(* IEC 61131-3 sources: Lasal/CPU_5344_V01/Class/generalMPScontrolSettings, 1 file *)

(* ---- generalMPScontrolSettings.st ---- *)
(*!
<Class
	Name               = "generalMPScontrolSettings"
	Revision           = "1.0"
	RealtimeTask       = "false"
	CyclicTask         = "false"
	BackgroundTask     = "false"
	Sigmatek           = "false"
	OSInterface        = "false"
	HighPriority       = "false"
	Automatic          = "false"
	UpdateMode         = "Prescan"
	SharedCommandTable = "true"
	Objectsize         = "(660,1080)">
	<Channels>
		<Server Name="addOutputOperations" Visualized="true" Initialize="true" WriteProtected="false" Retentive="false"/>
		<Server Name="amountOfUnits" Visualized="true" Initialize="true" DefValue="7" WriteProtected="false" Retentive="false"/>
		<Server Name="ClassSvr" Visualized="false" Initialize="false" WriteProtected="true" Retentive="false"/>
		<Server Name="combineOperations" Visualized="true" Initialize="true" DefValue="1" WriteProtected="false" Retentive="false"/>
		<Server Name="freeLoadDistance" Visualized="true" Initialize="false" WriteProtected="false" Retentive="false"/>
		<Server Name="gripDistanceInputWagon" Visualized="true" Initialize="false" WriteProtected="false" Retentive="false"/>
		<Server Name="lengthBetweenPieces" Visualized="true" Initialize="false" WriteProtected="false" Retentive="false"/>
		<Server Name="machineName" Class="StringRAM" Visualized="true" Remotely="true" Initialize="true" WriteProtected="false" Retentive="false"/>
		<Server Name="maxProductLength" Visualized="true" Initialize="true" WriteProtected="false" Retentive="false"/>
		<Server Name="maxScrapLength" Visualized="true" Initialize="false" WriteProtected="false" Retentive="false"/>
		<Server Name="maxTakeOverPos" Visualized="true" Initialize="false" WriteProtected="false" Retentive="false"/>
		<Server Name="minPosWagonUp" Visualized="true" Initialize="false" WriteProtected="false" Retentive="false"/>
		<Server Name="minProductLength" Visualized="true" Initialize="true" DefValue="1000" WriteProtected="false" Retentive="false"/>
		<Server Name="minScrapLengthEnd" Visualized="true" Initialize="false" WriteProtected="false" Retentive="false"/>
		<Server Name="minScrapLengthFront" Visualized="true" Initialize="false" WriteProtected="false" Retentive="false"/>
		<Server Name="minTakeOverPos" Visualized="true" Initialize="false" WriteProtected="false" Retentive="false"/>
		<Server Name="moveBigWasteToMagazine" Visualized="true" Initialize="false" WriteProtected="true" Retentive="false"/>
		<Server Name="moveToMinPosAfterProduction" Visualized="true" Initialize="true" DefValue="0" WriteProtected="false" Retentive="false"/>
		<Server Name="MPS_nr" Visualized="true" Initialize="true" DefValue="4444" WriteProtected="true" Retentive="false"/>
		<Server Name="noEndSaw" Visualized="true" Initialize="false" WriteProtected="false" Retentive="false"/>
		<Server Name="noFrontSaw" Visualized="true" Initialize="false" WriteProtected="false" Retentive="false"/>
		<Server Name="noWasteStop" Visualized="true" Initialize="false" WriteProtected="false" Retentive="false"/>
		<Server Name="optimumTakeOverPos" Visualized="true" Initialize="false" WriteProtected="false" Retentive="false"/>
		<Server Name="overtakeActive" Visualized="true" Initialize="false" WriteProtected="false" Retentive="false"/>
		<Server Name="turnPointSawAtOutputSide" Visualized="true" Initialize="false" WriteProtected="false" Retentive="false"/>
		<Server Name="wasteAtFront" Visualized="true" Initialize="false" WriteProtected="false" Retentive="false"/>
		<Server Name="wasteStopForEndWaste" Visualized="true" Initialize="false" WriteProtected="false" Retentive="false"/>
		<Server Name="yPosTurnPointSaw" Visualized="true" Initialize="false" WriteProtected="false" Retentive="false"/>
		<Client Name="ctrlCalc" Required="true" Internal="false"/>
		<Client Name="ctrlSettings" Required="true" Internal="false"/>
		<Client Name="iMaxPosWagon" Required="true" Internal="false"/>
		<Client Name="typeMachine" Required="true" Internal="true"/>
	</Channels>
	<Network Name="generalMPScontrolSettings">
		<!-- List of Components in this network -->
		<Components>
			<Object
				Name       = "typeMachine"
				Class      = "StringRAM"
				Position   = "(60,180)"
				Visualized = "true"
				Remotely   = "true">
				<Channels>
					<Server Name="Data"/>
					<Client Name="SingleRealloc" Value="1"/>
					<Client Name="UseFile"/>
				</Channels>
			</Object>
		</Components>
		<Comments>
		</Comments>
		<!-- List of Connections in this network -->
		<Connections>
			<Connection Source="this.typeMachine" Destination="typeMachine.Data"/>
			<Connection Source="this.machineName" Destination="typeMachine.Data" Vertices="(758,330),(586,270),"/>
		</Connections>
		<!-- Headerfiles -->
		<Options>
		</Options>
	</Network>
</Class>
*)
generalMPScontrolSettings : CLASS
  //Servers:
	ClassSvr 	: SvrChCmd_DINT;
	MPS_nr 	: SvrCh_DINT;
	machineName 	: SvrChCmd_UDINT;
	amountOfUnits 	: SvrCh_DINT;
	minProductLength 	: SvrCh_DINT;
	maxProductLength 	: SvrCh_DINT;
	minScrapLengthFront 	: SvrCh_DINT;
	minScrapLengthEnd 	: SvrCh_DINT;
	maxScrapLength 	: SvrCh_DINT;
	lengthBetweenPieces 	: SvrCh_DINT;
	freeLoadDistance 	: SvrCh_DINT;
	noFrontSaw 	: SvrCh_DINT;
	noEndSaw 	: SvrCh_DINT;
	wasteAtFront 	: SvrCh_DINT;
	turnPointSawAtOutputSide 	: SvrCh_DINT;
	yPosTurnPointSaw 	: SvrCh_DINT;
	moveToMinPosAfterProduction 	: SvrCh_DINT;
	gripDistanceInputWagon 	: SvrCh_DINT;
	moveBigWasteToMagazine 	: SvrCh_DINT;
	overtakeActive 	: SvrCh_DINT;
	combineOperations 	: SvrCh_DINT;
	noWasteStop 	: SvrCh_DINT;
	wasteStopForEndWaste 	: SvrCh_DINT;
	optimumTakeOverPos 	: SvrCh_DINT;
	minTakeOverPos 	: SvrCh_DINT;
	maxTakeOverPos 	: SvrCh_DINT;
	minPosWagonUp 	: SvrCh_DINT;
	addOutputOperations 	: SvrCh_DINT;
  //Clients:
	typeMachine 	: CltChCmd_StringRAM;
	ctrlSettings 	: CltChCmd_dbSettings;
	iMaxPosWagon 	: CltCh_DINT;
	ctrlCalc 	: CltChCmd_calcOperationListV2;
  //Variables:
  //Functions:

	FUNCTION VIRTUAL GLOBAL machineName::Read
		VAR_OUTPUT
			output (EAX) 	: UDINT;
		END_VAR;

	FUNCTION VIRTUAL GLOBAL machineName::Write
		VAR_INPUT
			input (EAX) 	: UDINT;
		END_VAR
		VAR_OUTPUT
			result (EAX) 	: UDINT;
		END_VAR;

	FUNCTION VIRTUAL GLOBAL maxProductLength::Read
		VAR_OUTPUT
			output (EAX) 	: DINT;
		END_VAR;

	FUNCTION VIRTUAL GLOBAL maxProductLength::Write
		VAR_INPUT
			input (EAX) 	: DINT;
		END_VAR
		VAR_OUTPUT
			result (EAX) 	: DINT;
		END_VAR;

	FUNCTION VIRTUAL GLOBAL minScrapLengthFront::Read
		VAR_OUTPUT
			output (EAX) 	: DINT;
		END_VAR;

	FUNCTION VIRTUAL GLOBAL minScrapLengthEnd::Read
		VAR_OUTPUT
			output (EAX) 	: DINT;
		END_VAR;

	FUNCTION VIRTUAL GLOBAL maxScrapLength::Read
		VAR_OUTPUT
			output (EAX) 	: DINT;
		END_VAR;

	FUNCTION VIRTUAL GLOBAL lengthBetweenPieces::Read
		VAR_OUTPUT
			output (EAX) 	: DINT;
		END_VAR;

	FUNCTION VIRTUAL GLOBAL freeLoadDistance::Read
		VAR_OUTPUT
			output (EAX) 	: DINT;
		END_VAR;

	FUNCTION VIRTUAL GLOBAL noFrontSaw::Read
		VAR_OUTPUT
			output (EAX) 	: DINT;
		END_VAR;

	FUNCTION VIRTUAL GLOBAL noEndSaw::Read
		VAR_OUTPUT
			output (EAX) 	: DINT;
		END_VAR;

	FUNCTION VIRTUAL GLOBAL wasteAtFront::Read
		VAR_OUTPUT
			output (EAX) 	: DINT;
		END_VAR;

	FUNCTION VIRTUAL GLOBAL turnPointSawAtOutputSide::Read
		VAR_OUTPUT
			output (EAX) 	: DINT;
		END_VAR;

	FUNCTION VIRTUAL GLOBAL yPosTurnPointSaw::Read
		VAR_OUTPUT
			output (EAX) 	: DINT;
		END_VAR;

	FUNCTION VIRTUAL GLOBAL moveToMinPosAfterProduction::Read
		VAR_OUTPUT
			output (EAX) 	: DINT;
		END_VAR;

	FUNCTION VIRTUAL GLOBAL gripDistanceInputWagon::Read
		VAR_OUTPUT
			output (EAX) 	: DINT;
		END_VAR;

	FUNCTION VIRTUAL GLOBAL moveBigWasteToMagazine::Read
		VAR_OUTPUT
			output (EAX) 	: DINT;
		END_VAR;

	FUNCTION VIRTUAL GLOBAL overtakeActive::Read
		VAR_OUTPUT
			output (EAX) 	: DINT;
		END_VAR;

	FUNCTION VIRTUAL GLOBAL noWasteStop::Read
		VAR_OUTPUT
			output (EAX) 	: DINT;
		END_VAR;

	FUNCTION VIRTUAL GLOBAL wasteStopForEndWaste::Read
		VAR_OUTPUT
			output (EAX) 	: DINT;
		END_VAR;

	FUNCTION VIRTUAL GLOBAL optimumTakeOverPos::Read
		VAR_OUTPUT
			output (EAX) 	: DINT;
		END_VAR;

	FUNCTION VIRTUAL GLOBAL minTakeOverPos::Read
		VAR_OUTPUT
			output (EAX) 	: DINT;
		END_VAR;

	FUNCTION VIRTUAL GLOBAL maxTakeOverPos::Read
		VAR_OUTPUT
			output (EAX) 	: DINT;
		END_VAR;

	FUNCTION VIRTUAL GLOBAL minPosWagonUp::Read
		VAR_OUTPUT
			output (EAX) 	: DINT;
		END_VAR;
  //Tables:
	FUNCTION @STD
		VAR_OUTPUT
			ret_code	: CONFSTATES;
		END_VAR;
	FUNCTION GLOBAL TAB @CT_;
END_CLASS;

#pragma using StringRAM
#pragma usingLtd calcOperationListV2
#pragma usingLtd dbSettings

// JdK 4-2-2020: generalMPScontrolSettings created for first test to read in settings to pc
// at this moment the class is only for storage off fixed machine data

FUNCTION VIRTUAL GLOBAL generalMPScontrolSettings::machineName::Read
	VAR_OUTPUT
		output (EAX) 	: UDINT;
	END_VAR

	machineName := typeMachine.Data.Read();
	output := machineName;

END_FUNCTION

FUNCTION VIRTUAL GLOBAL generalMPScontrolSettings::machineName::Write
	VAR_INPUT
		input (EAX) 	: UDINT;
	END_VAR
	VAR_OUTPUT
		result (EAX) 	: UDINT;
	END_VAR

	machineName := input;
	result := (typeMachine.Data.Write(machineName))$UDINT;

END_FUNCTION

FUNCTION VIRTUAL GLOBAL generalMPScontrolSettings::maxProductLength::Read
	VAR_OUTPUT
		output (EAX) 	: DINT;
	END_VAR

  iMaxPosWagon:= iMaxPosWagon.Read();
  maxProductLength:=iMaxPosWagon-ctrlSettings.offsetTakeIn-ctrlSettings.freeSpaceLoadMaterial;
	output := maxProductLength;

END_FUNCTION

FUNCTION VIRTUAL GLOBAL generalMPScontrolSettings::minScrapLengthFront::Read
	VAR_OUTPUT
		output (EAX) 	: DINT;
	END_VAR
  minScrapLengthFront:=ctrlSettings.minFrontWaste;
	output := minScrapLengthFront;

END_FUNCTION

FUNCTION VIRTUAL GLOBAL generalMPScontrolSettings::minScrapLengthEnd::Read
	VAR_OUTPUT
		output (EAX) 	: DINT;
	END_VAR
  minScrapLengthEnd:=ctrlSettings.minEndWaste;
	output := minScrapLengthEnd;

END_FUNCTION

FUNCTION VIRTUAL GLOBAL generalMPScontrolSettings::maxScrapLength::Read
	VAR_OUTPUT
		output (EAX) 	: DINT;
	END_VAR
  maxScrapLength:=ctrlSettings.maxLengthWaste;
	output := maxScrapLength;

END_FUNCTION

FUNCTION VIRTUAL GLOBAL generalMPScontrolSettings::freeLoadDistance::Read
	VAR_OUTPUT
		output (EAX) 	: DINT;
	END_VAR
  freeLoadDistance:=ctrlSettings.freeSpaceLoadMaterial;
	output := freeLoadDistance;

END_FUNCTION

FUNCTION VIRTUAL GLOBAL generalMPScontrolSettings::noFrontSaw::Read
	VAR_OUTPUT
		output (EAX) 	: DINT;
	END_VAR
  noFrontSaw:=ctrlSettings.doFrontWaste=0;//   .DoFrontWastePiece=0;
	output := noFrontSaw;

END_FUNCTION

FUNCTION VIRTUAL GLOBAL generalMPScontrolSettings::noEndSaw::Read
	VAR_OUTPUT
		output (EAX) 	: DINT;
	END_VAR
  noEndSaw:=ctrlSettings.DoEndWaste=0;
	output := noEndSaw;

END_FUNCTION

FUNCTION VIRTUAL GLOBAL generalMPScontrolSettings::wasteAtFront::Read
	VAR_OUTPUT
		output (EAX) 	: DINT;
	END_VAR
  wasteAtFront:=ctrlSettings.allWasteAtFront;
	output := wasteAtFront;

END_FUNCTION

FUNCTION VIRTUAL GLOBAL generalMPScontrolSettings::turnPointSawAtOutputSide::Read
	VAR_OUTPUT
		output (EAX) 	: DINT;
	END_VAR
  turnPointSawAtOutputSide:=ctrlCalc.sParTurnPointAtOutputSide;
	output := turnPointSawAtOutputSide;

END_FUNCTION

FUNCTION VIRTUAL GLOBAL generalMPScontrolSettings::yPosTurnPointSaw::Read
	VAR_OUTPUT
		output (EAX) 	: DINT;
	END_VAR
  yPosTurnPointSaw:=ctrlCalc.sParYposTurnPoint;
	output := yPosTurnPointSaw;

END_FUNCTION

FUNCTION VIRTUAL GLOBAL generalMPScontrolSettings::moveToMinPosAfterProduction::Read
	VAR_OUTPUT
		output (EAX) 	: DINT;
	END_VAR
  moveToMinPosAfterProduction:=ctrlCalc;
	output := moveToMinPosAfterProduction;

END_FUNCTION

FUNCTION VIRTUAL GLOBAL generalMPScontrolSettings::gripDistanceInputWagon::Read
	VAR_OUTPUT
		output (EAX) 	: DINT;
	END_VAR
  gripDistanceInputWagon:=ctrlSettings.lengthGripProfile;
	output := gripDistanceInputWagon;

END_FUNCTION

FUNCTION VIRTUAL GLOBAL generalMPScontrolSettings::moveBigWasteToMagazine::Read
	VAR_OUTPUT
		output (EAX) 	: DINT;
	END_VAR

  moveBigWasteToMagazine:= ctrlSettings.moveBigWasteToMagazin;
	output := moveBigWasteToMagazine;

END_FUNCTION

FUNCTION VIRTUAL GLOBAL generalMPScontrolSettings::overtakeActive::Read
	VAR_OUTPUT
		output (EAX) 	: DINT;
	END_VAR

  overtakeActive:= ctrlSettings.overTakeActive;
	output := overtakeActive;

END_FUNCTION

FUNCTION VIRTUAL GLOBAL generalMPScontrolSettings::noWasteStop::Read
	VAR_OUTPUT
		output (EAX) 	: DINT;
	END_VAR

  noWasteStop:= ctrlSettings.noWasteStop;
	output := noWasteStop;

END_FUNCTION

FUNCTION VIRTUAL GLOBAL generalMPScontrolSettings::wasteStopForEndWaste::Read
	VAR_OUTPUT
		output (EAX) 	: DINT;
	END_VAR

  wasteStopForEndWaste:= ctrlSettings.wasteStopForEndWaste & ctrlSettings.noWasteStop=0;
	output := wasteStopForEndWaste;

END_FUNCTION

FUNCTION VIRTUAL GLOBAL generalMPScontrolSettings::optimumTakeOverPos::Read
	VAR_OUTPUT
		output (EAX) 	: DINT;
	END_VAR

  optimumTakeOverPos:= ctrlSettings.optimumTakeOverPos;
	output := optimumTakeOverPos;

END_FUNCTION

FUNCTION VIRTUAL GLOBAL generalMPScontrolSettings::minTakeOverPos::Read
	VAR_OUTPUT
		output (EAX) 	: DINT;
	END_VAR

  minTakeOverPos:= ctrlSettings.minTakeOverPos;
	output := minTakeOverPos;

END_FUNCTION

FUNCTION VIRTUAL GLOBAL generalMPScontrolSettings::maxTakeOverPos::Read
	VAR_OUTPUT
		output (EAX) 	: DINT;
	END_VAR

  maxTakeOverPos:= ctrlSettings.maxTakeOverPos;
	output := maxTakeOverPos;

END_FUNCTION

FUNCTION VIRTUAL GLOBAL generalMPScontrolSettings::minPosWagonUp::Read
	VAR_OUTPUT
		output (EAX) 	: DINT;
	END_VAR

  minPosWagonUp:= ctrlSettings.minPosWagonUp;
	output := minPosWagonUp;

END_FUNCTION

FUNCTION VIRTUAL GLOBAL generalMPScontrolSettings::maxProductLength::Write
	VAR_INPUT
		input (EAX) 	: DINT;
	END_VAR
	VAR_OUTPUT
		result (EAX) 	: DINT;
	END_VAR

	maxProductLength := maxProductLength.Read();
	result := maxProductLength;

END_FUNCTION

FUNCTION VIRTUAL GLOBAL generalMPScontrolSettings::lengthBetweenPieces::Read
	VAR_OUTPUT
		output (EAX) 	: DINT;
	END_VAR

  lengthBetweenPieces:= ctrlSettings.lengthBetweenPiece;
	output := lengthBetweenPieces;

END_FUNCTION
